FUNCTION_BLOCK FB_AutomaticControl
VAR_INPUT
	bEnable								: BOOL;
	bStartMotion 						: BOOL;
	bStopMotion 						: BOOL;
	stValveOutputGeneratorSettings  	: ST_ValveOutputGeneratorSettings;
END_VAR
VAR_OUTPUT
	fTime : LREAL;
	fNormalizedValveOpeningRefSignal : LREAL;
END_VAR
VAR
	fbClock 					: FB_Clock;	
	fbValveOutputGenerator 		: FB_ValveOutputGenerator;	
END_VAR

fbClock(
	bStart := bStartMotion,
	bStop := bStopMotion,
	fCycleTime := G_Parameters.fCyclicTime
);

fbValveOutputGenerator(
	bEnable := bEnable,
	stValveOutputGeneratorSettings := stValveOutputGeneratorSettings,
	fClock_s := fbClock.fTime
);

fNormalizedValveOpeningRefSignal := fbValveOutputGenerator.fNormalizedValveOutputRef;

END_FUNCTION_BLOCK

(* stored: Version 1.1.0.1, ProductVersion 3.1.4024.11
   POU FB_AutomaticControl: Id {b543be1d-46f1-4ea5-ae35-9d7ea7728984}, SpecialFunc None *)
